PROGRAM MAIN
VAR
	rTemp :REAL;
END_VAR

END_PROGRAM

(* stored: Version 1.1.0.1, ProductVersion 3.1.4024.12
   POU MAIN: Id {3eed1957-7b5f-40df-a590-832bbf1d6005}, SpecialFunc None *)
